(* CoDeSys 2.3 export: IPADDRESS.EXP *)

(* Data type in STRUCT *)
TYPE IPAddress :
STRUCT
	length: Length;
	items: ARRAY [0..32767] OF BYTE;
END_STRUCT
END_TYPE
